// SIMATIC S7-200 project (STEP 7-Micro/WIN), CPU 224 CN REL 02.01

SYMBOL_TABLE 用户定义1
INI_CD           VW360    // 初始化密码
DEC_S            V0.0     // 圈数减标志位
ADD_S            V0.1     // 圈数加标志位
FWD              V0.2     // 长度正向增加
REV              V0.3     // 长度反向增加
sensor           V0.4     // 测速点
Q0_MODE          VW80
Q1_MODE          VW82
Q2_MODE          VW84
Q3_MODE          VW86
Q4_MODE          VW88
Q5_MODE          VW90
Q6_MODE          VW92
Q7_MODE          VW94
Q8_MODE          VW96
Q9_MODE          VW98
QS               VD10     // 圈数值
PULS_DI          VD14     // 脉冲数（双整型）
PULS_R           VD18     // 脉冲数（实数型）
CODE             VD22     // 码值
CODE_END         VD26     // 编码器最终生成值
GEAR             VD30     // 减速比
FIX_QT           VD34     // 修正系数
DIA              VD38     // 卷筒直径
GIRTH            VD42     // 周长
TO_LONG          VD46     // 转换为长度
BD_BUFFER        VD50     // 标定缓存
COLLATE          VD54     // 对比值
FIX_V            VD58     // 修正值
FIX_ACT          VD62     // 当前修正值
FIX_BUFFER       VD66     // 位置缓存
POSITION         VD70     // 当前位置
SPEED            VD76     // 运动速度
temp1            VD100
temp2            VD104    // 单圈长度
temp3            VD108
temp4            VD112
PST1             VD116    // 上次位置
speed0           VD120
speed1           VD124
speed2           VD128
speed3           VD132
temp5            VD136
temp6            VD140
temp7            VD144
DIA_REM          VD148
GEAR_REM         VD152
FIX_QT_REM       VD156
Q0_SET1          VD160
Q0_SET2          VD164
Q1_SET1          VD168
Q1_SET2          VD172
Q2_SET1          VD176
Q2_SET2          VD180
Q3_SET1          VD184
Q3_SET2          VD188
Q4_SET1          VD192
Q4_SET2          VD196
Q5_SET1          VD220
Q5_SET2          VD224
Q6_SET1          VD228
Q6_SET2          VD232
Q7_SET1          VD236
Q7_SET2          VD240
Q8_SET1          VD244
Q8_SET2          VD248
Q9_SET1          VD252
Q9_SET2          VD256
DIR_CACHE        VW74     // 方向修改码
END_SYMBOL_TABLE

SYMBOL_TABLE S7-200 符号
Always_On        SM0.0    // 始终接通为 ON
Clock_1s         SM0.5    // 在 1 秒钟的循环周期内，接通为 ON 0.5 秒，关断为 OFF 0.5  秒
END_SYMBOL_TABLE

ORGANIZATION_BLOCK 主程序:OB1
TITLE=程序注释
// 传送带通过格雷码转换子程序将编码器数据转换为二进制并计算圈数，再通过线性标定子程序使用减速比和修正系数转换为实际长度。前进方向命令或后退方向命令必须互斥，不能同时激活；若两者同时有效，系统将保持上一次位置不变，以防止传送带冲突移动导致设备损坏或位置计算错误。系统通过检测前进方向命令和后退方向命令的状态，确定传送带的运行方向。
// 基于当前位置，各站点如站0根据模式决定输出。模式0时，若位置小于站0设定值1则激活；模式1时，位置在设定值1和站0设定值2之间激活；模式2时，大于设定值1激活。所有设定值必须在用户按下F7后加载，确保操作安全且准确。
// 系统还计算运动速度基于位置变化，涉及多个临时变量，确保动态监控。显示控制根据模式显示状态，如模式0显示“小于值1”，便于操作员监控。用户通过按钮如F1-F8初始化参数或切换模式，必须经过去抖处理，避免误操作；系统启动时，始终接通标志确保所有标志初始化，防止未定义状态。
// 
BEGIN
Network 1
LD     Always_On:SM0.0
CALL   GRAY:SBR3
CALL   LINE:SBR0
CALL   PST:SBR4
CALL   CAM:SBR5
?000
Network 2 // 载入预设值1
LD     F7:V569.6
AW=    INI_CD:VW360, 20
LPS
MOVR   15.0, Q0_SET1:VD160
AENO
MOVR   17.5, Q1_SET1:VD168
AENO
MOVR   25.0, Q2_SET1:VD176
AENO
MOVR   105.0, Q3_SET1:VD184
AENO
MOVR   110.0, Q4_SET1:VD192
LRD
MOVR   0.0, Q0_SET2:VD164
AENO
MOVR   100.0, Q1_SET2:VD172
AENO
MOVR   90.0, Q2_SET2:VD180
AENO
MOVR   105.0, Q3_SET2:VD188
AENO
MOVR   110.0, Q4_SET2:VD196
LRD
MOVR   105.0, Q5_SET1:VD220
AENO
MOVR   20.0, Q6_SET1:VD228
AENO
MOVR   30.0, Q7_SET1:VD236
AENO
MOVR   15.0, Q8_SET1:VD244
AENO
MOVR   10.0, Q9_SET1:VD252
LPP
MOVR   105.0, Q5_SET2:VD224
AENO
MOVR   102.5, Q6_SET2:VD232
AENO
MOVR   95.0, Q7_SET2:VD240
AENO
MOVR   0.0, Q8_SET2:VD248
AENO
MOVR   0.0, Q9_SET2:VD256
Network 3 // 载入预设值2
LD     F7:V569.6
AW=    INI_CD:VW360, 20
LPS
MOVR   5.0, GEAR:VD30
AENO
MOVR   1.0, FIX_QT:VD34
AENO
MOVR   1.25, DIA:VD38
AENO
MOVR   DIA:VD38, GIRTH:VD42
AENO
*R     3.141593, GIRTH:VD42
AENO
MOVR   GIRTH:VD42, temp1:VD100
AENO
*R     GEAR:VD30, temp1:VD100
AENO
MOVR   temp1:VD100, temp2:VD104
*R     FIX_QT:VD34, temp2:VD104
LRD
MOVR   DIA:VD38, DIA_REM:VD148
AENO
MOVR   GEAR:VD30, GEAR_REM:VD152
AENO
MOVR   FIX_QT:VD34, FIX_QT_REM:VD156
AENO
SCPY   "已生效", VB210
AENO
MOVW   0, INI_CD:VW360
LRD
MOVW   0, Q0_MODE:VW80
AENO
MOVW   1, Q1_MODE:VW82
AENO
MOVW   1, Q2_MODE:VW84
AENO
MOVW   2, Q3_MODE:VW86
AENO
MOVW   2, Q4_MODE:VW88
LPP
MOVW   2, Q5_MODE:VW90
AENO
MOVW   1, Q6_MODE:VW92
AENO
MOVW   1, Q7_MODE:VW94
AENO
MOVW   0, Q8_MODE:VW96
AENO
MOVW   0, Q9_MODE:VW98
Network 4
LD     F1:V569.0
EU
LPS
AN     M10.1
S      M10.0, 1
LPP
A      M10.1
R      M10.0, 1
Network 5
LD     M10.0
=      M10.1
Network 6
LD     F2:V569.1
S      M10.2, 1
R      M10.3, 1
Network 7
LD     F3:V569.2
S      M10.3, 1
R      M10.2, 1
Network 8
LD     M10.0
A      M10.2
A      M10.4
+I     1, MW4
Network 9
LD     M10.0
A      M10.3
A      M10.4
+I     -1, MW4
Network 10
LDN    M10.4
TON    T36, 2
Network 11
LD     T36
=      M10.4
Network 12
LD     Always_On:SM0.0
MOVB   MB5, MB6
AENO
SRB    MB6, 1
AENO
MOVB   MB5, MB8
AENO
INVB   MB8
AENO
MOVB   MB6, MB9
INVB   MB9
Network 13
LD     Always_On:SM0.0
MOVB   MB5, MB12
AENO
ANDB   MB9, MB12
AENO
MOVB   MB6, MB13
AENO
ANDB   MB8, MB13
AENO
MOVB   MB12, MB7
ORB    MB13, MB7
END_ORGANIZATION_BLOCK

SUBROUTINE_BLOCK LINE:SBR0
TITLE=线性标定
// 将编码器的圈数值转换成长度值
BEGIN
Network 1
LDR=   GEAR:VD30, 0.0
MOVR   1.0, GEAR:VD30
Network 2
LDR=   FIX_QT:VD34, 0.0
MOVR   1.0, FIX_QT:VD34
Network 3
LD     F5:V569.4
EU
LPS
MOVR   DIA:VD38, GIRTH:VD42
AENO
*R     3.141593, GIRTH:VD42
AENO
MOVR   GIRTH:VD42, temp1:VD100
AENO
*R     GEAR:VD30, temp1:VD100
AENO
MOVR   temp1:VD100, temp2:VD104
AENO
*R     FIX_QT:VD34, temp2:VD104
AENO
SCPY   "已生效", VB210
LPP
MOVR   DIA:VD38, DIA_REM:VD148
AENO
MOVR   GEAR:VD30, GEAR_REM:VD152
AENO
MOVR   FIX_QT:VD34, FIX_QT_REM:VD156
Network 4
LDR<>  DIA:VD38, DIA_REM:VD148
OR<>   GEAR:VD30, GEAR_REM:VD152
OR<>   FIX_QT:VD34, FIX_QT_REM:VD156
SCPY   "未生效", VB210
Network 5
LD     Always_On:SM0.0
MOVR   temp2:VD104, TO_LONG:VD46
*R     CODE_END:VD26, TO_LONG:VD46
MOVR   TO_LONG:VD46, COLLATE:VD54
-R     BD_BUFFER:VD50, COLLATE:VD54
Network 6
LD     F5:V569.4
EU
MOVR   TO_LONG:VD46, BD_BUFFER:VD50
END_SUBROUTINE_BLOCK

// SBR1: protected block, not included

// SBR2: protected block, not included

SUBROUTINE_BLOCK GRAY:SBR3
TITLE=格雷码转换
// 将格雷码值转换为2进制，最后转换为圈数
BEGIN
Network 1 // 网络标题
// 网络注释
LD     M7.7
=      M1.7
Network 2
LD     M1.7
AN     M7.6
LDN    M1.7
A      M7.6
OLD
=      M1.6
Network 3
LD     M1.6
AN     M7.5
LDN    M1.6
A      M7.5
OLD
=      M1.5
Network 4
LD     M1.5
AN     M7.4
LDN    M1.5
A      M7.4
OLD
=      M1.4
Network 5
LD     M1.4
AN     M7.3
LDN    M1.4
A      M7.3
OLD
=      M1.3
Network 6
LD     M1.3
AN     M7.2
LDN    M1.3
A      M7.2
OLD
=      M1.2
Network 7
LD     M1.2
AN     M7.1
LDN    M1.2
A      M7.1
OLD
=      M1.1
Network 8
LD     M1.1
AN     M7.0
LDN    M1.1
A      M7.0
OLD
=      M1.0
Network 9
LD     Always_On:SM0.0
MOVB   0, MB0
Network 10 // 圈计数减标记
LDW<=  MW0, 30
S      DEC_S:V0.0, 1
Network 11 // 圈计数加标记
LDW>=  MW0, 225
S      ADD_S:V0.1, 1
Network 12
LDW>   MW0, 30
AW<    MW0, 225
R      DEC_S:V0.0, 1
R      ADD_S:V0.1, 1
Network 13 // 增加圈
LD     ADD_S:V0.1
AW<=   MW0, 30
+R     256.0, QS:VD10
AENO
R      ADD_S:V0.1, 1
Network 14 // 减少圈
LD     DEC_S:V0.0
AW>=   MW0, 225
+R     -256.0, QS:VD10
AENO
R      DEC_S:V0.0, 1
Network 15 // 编码值生成
LD     Always_On:SM0.0
ITD    MW0, PULS_DI:VD14
AENO
DTR    PULS_DI:VD14, PULS_R:VD18
AENO
MOVR   QS:VD10, CODE:VD22
+R     PULS_R:VD18, CODE:VD22
Network 16
LD     Always_On:SM0.0
MOVR   CODE:VD22, CODE_END:VD26
/R     256.0, CODE_END:VD26
END_SUBROUTINE_BLOCK

SUBROUTINE_BLOCK PST:SBR4
TITLE=位置生成
// 
BEGIN
Network 1 // 网络标题
// 网络注释
LDR<>  FIX_V:VD58, FIX_ACT:VD62
A      F8:V569.7
TON    T37, 30
Network 2
LD     T37
EU
MOVR   FIX_V:VD58, FIX_ACT:VD62
AENO
MOVR   TO_LONG:VD46, FIX_BUFFER:VD66
Network 3
LD     FWD:V0.2
AN     REV:V0.3
MOVR   TO_LONG:VD46, temp3:VD108
AENO
-R     FIX_BUFFER:VD66, temp3:VD108
AENO
MOVR   FIX_ACT:VD62, POSITION:VD70
AENO
+R     temp3:VD108, POSITION:VD70
AENO
SCPY   "正逻辑", VB200
Network 4
LDN    FWD:V0.2
A      REV:V0.3
MOVR   TO_LONG:VD46, temp3:VD108
AENO
-R     FIX_BUFFER:VD66, temp3:VD108
AENO
MOVR   FIX_ACT:VD62, POSITION:VD70
AENO
-R     temp3:VD108, POSITION:VD70
AENO
SCPY   "负逻辑", VB200
Network 5
LDN    FWD:V0.2
AN     REV:V0.3
LD     FWD:V0.2
A      REV:V0.3
OLD
TON    T38, 20
Network 6
LD     T38
S      FWD:V0.2, 1
Network 7
LDW=   DIR_CACHE:VW74, 15
A      F6:V569.5
A      FWD:V0.2
R      FWD:V0.2, 1
S      REV:V0.3, 1
MOVW   0, DIR_CACHE:VW74
Network 8
LDW=   DIR_CACHE:VW74, 15
A      F6:V569.5
A      REV:V0.3
R      REV:V0.3, 1
S      FWD:V0.2, 1
MOVW   0, DIR_CACHE:VW74
Network 9 // 测速
LDN    sensor:V0.4
TON    T33, 10
Network 10
LD     T33
=      sensor:V0.4
Network 11
LD     sensor:V0.4
LPS
MOVR   POSITION:VD70, temp4:VD112
AENO
-R     PST1:VD116, temp4:VD112
AENO
MOVR   POSITION:VD70, PST1:VD116
AENO
MOVR   speed2:VD128, speed3:VD132
AENO
MOVR   speed1:VD124, speed2:VD128
AENO
MOVR   speed0:VD120, speed1:VD124
AENO
MOVR   temp4:VD112, speed0:VD120
*R     10.0, speed0:VD120
LPP
MOVR   speed0:VD120, temp5:VD136
AENO
+R     speed1:VD124, temp5:VD136
AENO
MOVR   speed2:VD128, temp6:VD140
AENO
+R     speed3:VD132, temp6:VD140
AENO
MOVR   temp5:VD136, temp7:VD144
AENO
+R     temp6:VD140, temp7:VD144
AENO
MOVR   temp7:VD144, SPEED:VD76
/R     4.0, SPEED:VD76
END_SUBROUTINE_BLOCK

SUBROUTINE_BLOCK CAM:SBR5
TITLE=子程序注释
BEGIN
Network 1 // 网络标题
// 网络注释
LDW>   Q0_MODE:VW80, 2
MOVW   0, Q0_MODE:VW80
Network 2 // 网络标题
// 网络注释
LDW>   Q1_MODE:VW82, 2
MOVW   0, Q1_MODE:VW82
Network 3 // 网络标题
// 网络注释
LDW>   Q2_MODE:VW84, 2
MOVW   0, Q2_MODE:VW84
Network 4 // 网络标题
// 网络注释
LDW>   Q3_MODE:VW86, 2
MOVW   0, Q3_MODE:VW86
Network 5 // 网络标题
// 网络注释
LDW>   Q4_MODE:VW88, 2
MOVW   0, Q4_MODE:VW88
Network 6 // 网络标题
// 网络注释
LDW>   Q5_MODE:VW90, 2
MOVW   0, Q5_MODE:VW90
Network 7 // 网络标题
// 网络注释
LDW>   Q6_MODE:VW92, 2
MOVW   0, Q6_MODE:VW92
Network 8 // 网络标题
// 网络注释
LDW>   Q7_MODE:VW94, 2
MOVW   0, Q7_MODE:VW94
Network 9 // 网络标题
// 网络注释
LDW>   Q8_MODE:VW96, 2
MOVW   0, Q8_MODE:VW96
Network 10 // 网络标题
// 网络注释
LDW>   Q9_MODE:VW98, 2
MOVW   0, Q9_MODE:VW98
Network 11
LDW=   Q0_MODE:VW80, 0
AR<=   POSITION:VD70, Q0_SET1:VD160
LDW=   Q0_MODE:VW80, 1
AR>    POSITION:VD70, Q0_SET1:VD160
AR<    POSITION:VD70, Q0_SET2:VD164
OLD
LDW=   Q0_MODE:VW80, 2
AR>=   POSITION:VD70, Q0_SET1:VD160
OLD
=      Q0.0
Network 12
LDW=   Q1_MODE:VW82, 0
AR<=   POSITION:VD70, Q1_SET1:VD168
LDW=   Q1_MODE:VW82, 1
AR>    POSITION:VD70, Q1_SET1:VD168
AR<    POSITION:VD70, Q1_SET2:VD172
OLD
LDW=   Q1_MODE:VW82, 2
AR>=   POSITION:VD70, Q1_SET1:VD168
OLD
=      Q0.1
Network 13
LDW=   Q2_MODE:VW84, 0
AR<=   POSITION:VD70, Q2_SET1:VD176
LDW=   Q2_MODE:VW84, 1
AR>    POSITION:VD70, Q2_SET1:VD176
AR<    POSITION:VD70, Q2_SET2:VD180
OLD
LDW=   Q2_MODE:VW84, 2
AR>=   POSITION:VD70, Q2_SET1:VD176
OLD
=      Q0.2
Network 14
LDW=   Q3_MODE:VW86, 0
AR<=   POSITION:VD70, Q3_SET1:VD184
LDW=   Q3_MODE:VW86, 1
AR>    POSITION:VD70, Q3_SET1:VD184
AR<    POSITION:VD70, Q3_SET2:VD188
OLD
LDW=   Q3_MODE:VW86, 2
AR>=   POSITION:VD70, Q3_SET1:VD184
OLD
=      Q0.3
Network 15
LDW=   Q4_MODE:VW88, 0
AR<=   POSITION:VD70, Q4_SET1:VD192
LDW=   Q4_MODE:VW88, 1
AR>    POSITION:VD70, Q4_SET1:VD192
AR<    POSITION:VD70, Q4_SET2:VD196
OLD
LDW=   Q4_MODE:VW88, 2
AR>=   POSITION:VD70, Q4_SET1:VD192
OLD
=      Q0.4
Network 16
LDW=   Q5_MODE:VW90, 0
AR<=   POSITION:VD70, Q5_SET1:VD220
LDW=   Q5_MODE:VW90, 1
AR>    POSITION:VD70, Q5_SET1:VD220
AR<    POSITION:VD70, Q5_SET2:VD224
OLD
LDW=   Q5_MODE:VW90, 2
AR>=   POSITION:VD70, Q5_SET1:VD220
OLD
=      Q0.5
Network 17
LDW=   Q6_MODE:VW92, 0
AR<=   POSITION:VD70, Q6_SET1:VD228
LDW=   Q6_MODE:VW92, 1
AR>    POSITION:VD70, Q6_SET1:VD228
AR<    POSITION:VD70, Q6_SET2:VD232
OLD
LDW=   Q6_MODE:VW92, 2
AR>=   POSITION:VD70, Q6_SET1:VD228
OLD
=      Q0.6
Network 18
LDW=   Q7_MODE:VW94, 0
AR<=   POSITION:VD70, Q7_SET1:VD236
LDW=   Q7_MODE:VW94, 1
AR>    POSITION:VD70, Q7_SET1:VD236
AR<    POSITION:VD70, Q7_SET2:VD240
OLD
LDW=   Q7_MODE:VW94, 2
AR>=   POSITION:VD70, Q7_SET1:VD236
OLD
=      Q0.7
Network 19
LDW=   Q8_MODE:VW96, 0
AR<=   POSITION:VD70, Q8_SET1:VD244
LDW=   Q8_MODE:VW96, 1
AR>    POSITION:VD70, Q8_SET1:VD244
AR<    POSITION:VD70, Q8_SET2:VD248
OLD
LDW=   Q8_MODE:VW96, 2
AR>=   POSITION:VD70, Q8_SET1:VD244
OLD
=      Q1.0
Network 20
LDW=   Q9_MODE:VW98, 0
AR<=   POSITION:VD70, Q9_SET1:VD252
LDW=   Q9_MODE:VW98, 1
AR>    POSITION:VD70, Q9_SET1:VD252
AR<    POSITION:VD70, Q9_SET2:VD256
OLD
LDW=   Q9_MODE:VW98, 2
AR>=   POSITION:VD70, Q9_SET1:VD252
OLD
=      Q1.1
Network 21
LD     Clock_1s:SM0.5
EU
CALL   DSP:SBR6
END_SUBROUTINE_BLOCK

SUBROUTINE_BLOCK DSP:SBR6
TITLE=子程序注释
BEGIN
Network 1 // 网络标题
// 网络注释
LDW=   Q0_MODE:VW80, 0
SCPY   "小于值1", VB260
Network 2 // 网络标题
// 网络注释
LDW=   Q0_MODE:VW80, 1
SCPY   "两值之间", VB260
Network 3 // 网络标题
// 网络注释
LDW=   Q0_MODE:VW80, 2
SCPY   "大于值1", VB260
Network 4 // 网络标题
// 网络注释
LDW=   Q1_MODE:VW82, 0
SCPY   "小于值1", VB270
Network 5 // 网络标题
// 网络注释
LDW=   Q1_MODE:VW82, 1
SCPY   "两值之间", VB270
Network 6 // 网络标题
// 网络注释
LDW=   Q1_MODE:VW82, 2
SCPY   "大于值1", VB270
Network 7 // 网络标题
// 网络注释
LDW=   Q2_MODE:VW84, 0
SCPY   "小于值1", VB280
Network 8 // 网络标题
// 网络注释
LDW=   Q2_MODE:VW84, 1
SCPY   "两值之间", VB280
Network 9 // 网络标题
// 网络注释
LDW=   Q2_MODE:VW84, 2
SCPY   "大于值1", VB280
Network 10 // 网络标题
// 网络注释
LDW=   Q3_MODE:VW86, 0
SCPY   "小于值1", VB290
Network 11 // 网络标题
// 网络注释
LDW=   Q3_MODE:VW86, 1
SCPY   "两值之间", VB290
Network 12 // 网络标题
// 网络注释
LDW=   Q3_MODE:VW86, 2
SCPY   "大于值1", VB290
Network 13 // 网络标题
// 网络注释
LDW=   Q4_MODE:VW88, 0
SCPY   "小于值1", VB300
Network 14 // 网络标题
// 网络注释
LDW=   Q4_MODE:VW88, 1
SCPY   "两值之间", VB300
Network 15 // 网络标题
// 网络注释
LDW=   Q4_MODE:VW88, 2
SCPY   "大于值1", VB300
Network 16 // 网络标题
// 网络注释
LDW=   Q5_MODE:VW90, 0
SCPY   "小于值1", VB310
Network 17 // 网络标题
// 网络注释
LDW=   Q5_MODE:VW90, 1
SCPY   "两值之间", VB310
Network 18 // 网络标题
// 网络注释
LDW=   Q5_MODE:VW90, 2
SCPY   "大于值1", VB310
Network 19 // 网络标题
// 网络注释
LDW=   Q6_MODE:VW92, 0
SCPY   "小于值1", VB320
Network 20 // 网络标题
// 网络注释
LDW=   Q6_MODE:VW92, 1
SCPY   "两值之间", VB320
Network 21 // 网络标题
// 网络注释
LDW=   Q6_MODE:VW92, 2
SCPY   "大于值1", VB320
Network 22 // 网络标题
// 网络注释
LDW=   Q7_MODE:VW94, 0
SCPY   "小于值1", VB330
Network 23 // 网络标题
// 网络注释
LDW=   Q7_MODE:VW94, 1
SCPY   "两值之间", VB330
Network 24 // 网络标题
// 网络注释
LDW=   Q7_MODE:VW94, 2
SCPY   "大于值1", VB330
Network 25 // 网络标题
// 网络注释
LDW=   Q8_MODE:VW96, 0
SCPY   "小于值1", VB340
Network 26 // 网络标题
// 网络注释
LDW=   Q8_MODE:VW96, 1
SCPY   "两值之间", VB340
Network 27 // 网络标题
// 网络注释
LDW=   Q8_MODE:VW96, 2
SCPY   "大于值1", VB340
Network 28 // 网络标题
// 网络注释
LDW=   Q9_MODE:VW98, 0
SCPY   "小于值1", VB350
Network 29 // 网络标题
// 网络注释
LDW=   Q9_MODE:VW98, 1
SCPY   "两值之间", VB350
Network 30 // 网络标题
// 网络注释
LDW=   Q9_MODE:VW98, 2
SCPY   "大于值1", VB350
END_SUBROUTINE_BLOCK

// (further data pages could not be read)
